// TIA Portal project "Practica_8_v2" (V14)

(* hardware
DEVICE "S7-1200 station_1"  S7-1200 Station
   slot 0: "Rack_0"  S7-1200 Rack  Rack  V1.0
   slot 1: "PLC_1"  CPU 1214C AC/DC/Rly  6ES7 214-1BG40-0XB0  V4.2
*)

// ===== PLC "PLC_1"  CPU 1214C AC/DC/Rly =====

VAR_GLOBAL   // PLC tag table "Default tag table"
   "PM" AT %I0.0 : Bool;
   "PP" AT %I0.1 : Bool;
   "FCA_1" AT %I0.2 : Bool;
   "FCB_1" AT %I0.3 : Bool;
   "CW_1" AT %Q0.0 : Bool;
   "CCW_1" AT %Q0.1 : Bool;
   "ENABLE" AT %M0.0 : Bool;
END_VAR

DATA_BLOCK "carrito_1"   // DB1
{ S7_Optimized_Access := 'TRUE' }
VERSION : 0.1
// stored: InstanceOfName carrito
"carrito"
BEGIN
END_DATA_BLOCK

DATA_BLOCK "CARROS"   // DB2
{ S7_Optimized_Access := 'TRUE' }
VERSION : 0.1
   VAR
      TE_CARRO1 : Time := T#10s;
      N_CARRO1 : Int := 5;
      TE_CARRO2 : Time := T#4s;
      N_CARRO2 : Int := 4;
   END_VAR
BEGIN
END_DATA_BLOCK

FUNCTION_BLOCK "carrito"   // FB1, LAD
{ S7_Optimized_Access := 'TRUE' }
VERSION : 0.1
   VAR_INPUT
      ENABLE : Bool;
      FCA : Bool;
      FCB : Bool;
      N : Int := 5;
      TE : Time := T#10s;
   END_VAR
   VAR_OUTPUT
      CW : Bool;
      CCW : Bool;
   END_VAR
   VAR
      ST_OFF : Bool;
      M1 : Bool := false;
      M2 : Bool;
      ST_M1 : Bool;
      ST_M2 : Bool;
      ST_A : Bool;
      ST_B : Bool;
   END_VAR
   VAR RETAIN
      CNT : CTU_INT;
   END_VAR
   VAR
      TIMER_B : TON_TIME;
      TIMER_A : TON_TIME;
   END_VAR
   VAR CONSTANT
      TA : Time := T#1s;
   END_VAR
   VAR_TEMP   // added for the SCL form of the ladder/FBD networks
      _w1 : Bool;
   END_VAR
   // CNT.PV := 0;
BEGIN

REGION Network 1
   // Inicialización.
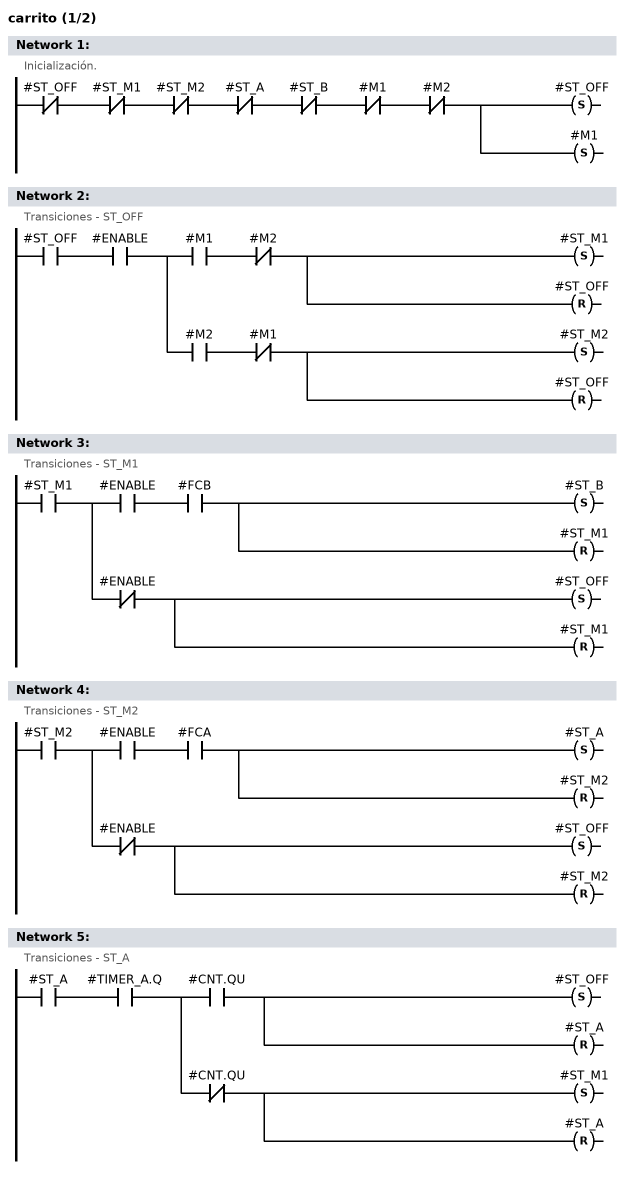
   RUNG wire#powerrail
      I_Contact( #ST_OFF )
      I_Contact( #ST_M1 )
      I_Contact( #ST_M2 )
      I_Contact( #ST_A )
      I_Contact( #ST_B )
      I_Contact( #M1 )
      I_Contact( #M2 )
      wire#w1
      S_Coil( #ST_OFF )
   END_RUNG
   RUNG wire#w1
      S_Coil( #M1 )
   END_RUNG
   // the same network as SCL:
   #_w1 := NOT #ST_OFF AND NOT #ST_M1 AND NOT #ST_M2 AND NOT #ST_A AND NOT #ST_B AND NOT #M1 AND NOT #M2;
   IF #_w1 THEN
       #ST_OFF := TRUE;
       #M1 := TRUE;
   END_IF;
END_REGION

REGION Network 2
   // Transiciones - ST_OFF
   RUNG wire#powerrail
      Contact( #ST_OFF )
      Contact( #ENABLE )
      wire#w1
      Contact( #M1 )
      I_Contact( #M2 )
      wire#w2
      S_Coil( #ST_M1 )
   END_RUNG
   RUNG wire#w2
      R_Coil( #ST_OFF )
   END_RUNG
   RUNG wire#w1
      Contact( #M2 )
      I_Contact( #M1 )
      wire#w3
      S_Coil( #ST_M2 )
   END_RUNG
   RUNG wire#w3
      R_Coil( #ST_OFF )
   END_RUNG
   // the same network as SCL:
   #_w1 := #ST_OFF AND #ENABLE;
   IF #_w1 AND #M1 AND NOT #M2 THEN
       #ST_M1 := TRUE;
       #ST_OFF := FALSE;
   END_IF;
   IF #_w1 AND #M2 AND NOT #M1 THEN
       #ST_M2 := TRUE;
       #ST_OFF := FALSE;
   END_IF;
END_REGION

REGION Network 3
   // Transiciones - ST_M1
   RUNG wire#powerrail
      Contact( #ST_M1 )
      wire#w1
      Contact( #ENABLE )
      Contact( #FCB )
      wire#w2
      S_Coil( #ST_B )
   END_RUNG
   RUNG wire#w2
      R_Coil( #ST_M1 )
   END_RUNG
   RUNG wire#w1
      I_Contact( #ENABLE )
      wire#w3
      S_Coil( #ST_OFF )
   END_RUNG
   RUNG wire#w3
      R_Coil( #ST_M1 )
   END_RUNG
   // the same network as SCL:
   IF #ST_M1 AND #ENABLE AND #FCB THEN #ST_B := TRUE; END_IF;
   #_w1 := #ST_M1;
   IF #ST_M1 AND #ENABLE AND #FCB THEN #ST_M1 := FALSE; END_IF;
   IF #_w1 AND NOT #ENABLE THEN
       #ST_OFF := TRUE;
       #ST_M1 := FALSE;
   END_IF;
END_REGION

REGION Network 4
   // Transiciones - ST_M2
   RUNG wire#powerrail
      Contact( #ST_M2 )
      wire#w1
      Contact( #ENABLE )
      Contact( #FCA )
      wire#w2
      S_Coil( #ST_A )
   END_RUNG
   RUNG wire#w2
      R_Coil( #ST_M2 )
   END_RUNG
   RUNG wire#w1
      I_Contact( #ENABLE )
      wire#w3
      S_Coil( #ST_OFF )
   END_RUNG
   RUNG wire#w3
      R_Coil( #ST_M2 )
   END_RUNG
   // the same network as SCL:
   IF #ST_M2 AND #ENABLE AND #FCA THEN #ST_A := TRUE; END_IF;
   #_w1 := #ST_M2;
   IF #ST_M2 AND #ENABLE AND #FCA THEN #ST_M2 := FALSE; END_IF;
   IF #_w1 AND NOT #ENABLE THEN
       #ST_OFF := TRUE;
       #ST_M2 := FALSE;
   END_IF;
END_REGION

REGION Network 5
   // Transiciones - ST_A
   RUNG wire#powerrail
      Contact( #ST_A )
      Contact( #TIMER_A.Q )
      wire#w1
      Contact( #CNT.QU )
      wire#w2
      S_Coil( #ST_OFF )
   END_RUNG
   RUNG wire#w2
      R_Coil( #ST_A )
   END_RUNG
   RUNG wire#w1
      I_Contact( #CNT.QU )
      wire#w3
      S_Coil( #ST_M1 )
   END_RUNG
   RUNG wire#w3
      R_Coil( #ST_A )
   END_RUNG
   // the same network as SCL:
   #_w1 := #ST_A AND #TIMER_A.Q;
   IF #_w1 AND #CNT.QU THEN
       #ST_OFF := TRUE;
       #ST_A := FALSE;
   END_IF;
   IF #_w1 AND NOT #CNT.QU THEN
       #ST_M1 := TRUE;
       #ST_A := FALSE;
   END_IF;
END_REGION

REGION Network 6
   // Transiciones - ST_B
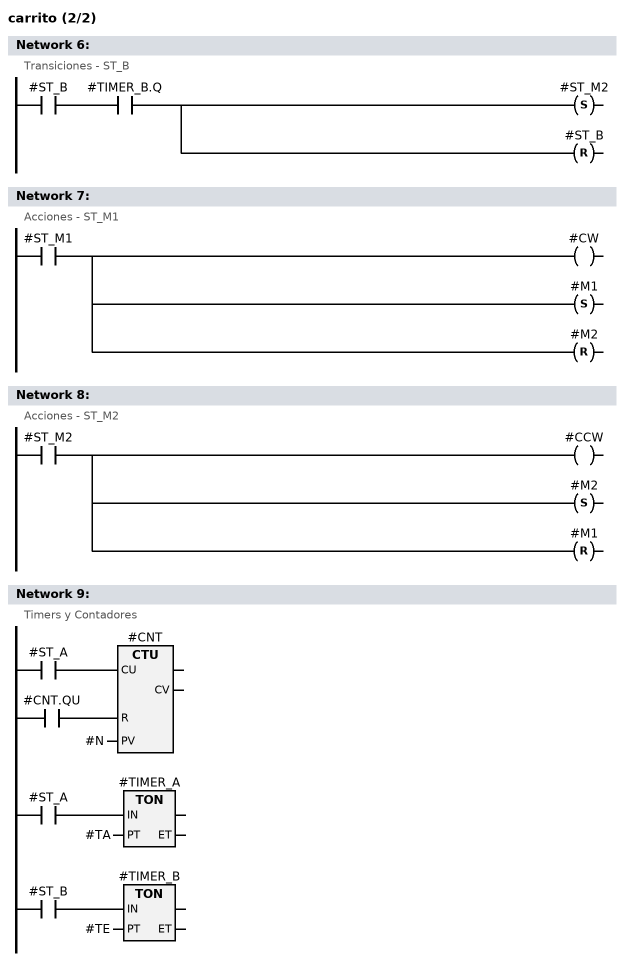
   RUNG wire#powerrail
      Contact( #ST_B )
      Contact( #TIMER_B.Q )
      wire#w1
      S_Coil( #ST_M2 )
   END_RUNG
   RUNG wire#w1
      R_Coil( #ST_B )
   END_RUNG
   // the same network as SCL:
   IF #ST_B AND #TIMER_B.Q THEN
       #ST_M2 := TRUE;
       #ST_B := FALSE;
   END_IF;
END_REGION

REGION Network 7
   // Acciones - ST_M1
   RUNG wire#powerrail
      Contact( #ST_M1 )
      wire#w1
      Coil( #CW )
   END_RUNG
   RUNG wire#w1
      S_Coil( #M1 )
   END_RUNG
   RUNG wire#w1
      R_Coil( #M2 )
   END_RUNG
   // the same network as SCL:
   #CW := #ST_M1;
   IF #ST_M1 THEN
       #M1 := TRUE;
       #M2 := FALSE;
   END_IF;
END_REGION

REGION Network 8
   // Acciones - ST_M2
   RUNG wire#powerrail
      Contact( #ST_M2 )
      wire#w1
      Coil( #CCW )
   END_RUNG
   RUNG wire#w1
      S_Coil( #M2 )
   END_RUNG
   RUNG wire#w1
      R_Coil( #M1 )
   END_RUNG
   // the same network as SCL:
   #CCW := #ST_M2;
   IF #ST_M2 THEN
       #M2 := TRUE;
       #M1 := FALSE;
   END_IF;
END_REGION

REGION Network 9
   // Timers y Contadores
   #CNT(CU := #ST_A, R := #CNT.QU, PV := #N);   // CTU
   #TIMER_A(IN := #ST_A, PT := #TA);   // TON
   #TIMER_B(IN := #ST_B, PT := #TE);   // TON
END_REGION
END_FUNCTION_BLOCK

ORGANIZATION_BLOCK "Main"   // OB1, LAD, ProgramCycle
TITLE = "Main Program Sweep (Cycle)"
{ S7_Optimized_Access := 'TRUE' }
VERSION : 0.1
   VAR_INPUT
      Initial_Call : Bool;   // Initial call of this OB
      Remanence : Bool;   // =True, if remanent data are available
   END_VAR
BEGIN

REGION Network 1
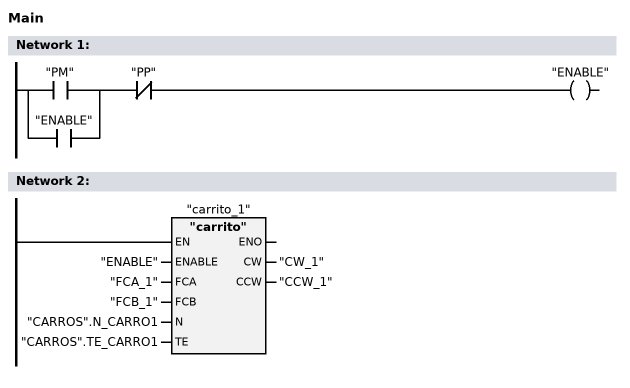
   RUNG wire#powerrail
      Contact( "PM" )
      wire#w1
      I_Contact( "PP" )
      Coil( "ENABLE" )
   END_RUNG
   RUNG wire#powerrail
      Contact( "ENABLE" )
   END_RUNG wire#w1
   // the same network as SCL:
   "ENABLE" := ("PM" OR "ENABLE") AND NOT "PP";
END_REGION

REGION Network 2
   RUNG wire#powerrail
      "carrito_1"(ENABLE := "ENABLE", FCA := "FCA_1", FCB := "FCB_1", N := "CARROS".N_CARRO1, TE := "CARROS".TE_CARRO1, CW => "CW_1", CCW => "CCW_1")
   END_RUNG
   // the same network as SCL:
   "carrito_1"(ENABLE := "ENABLE",   // "carrito"
               FCA := "FCA_1",
               FCB := "FCB_1",
               N := "CARROS".N_CARRO1,
               TE := "CARROS".TE_CARRO1,
               CW => "CW_1",
               CCW => "CCW_1");
END_REGION
END_ORGANIZATION_BLOCK